TYPE ST_CX_AMSAddress :
STRUCT
	arrAMSNetID			: AMSNETID;
	nPortNo				: UINT;
END_STRUCT
END_TYPE

(* stored: Version 1.1.0.1, ProductVersion 3.1.4024.15
   DUT ST_CX_AMSAddress: Id {fb3c9cf6-d752-4f82-aef5-75525c2f4e18} *)
